{attribute 'GeneratedUsingTerminal: EL3773-0000-0019'}
{attribute addProperty BoxType "EL3773-0000-0019"}
{attribute addProperty Id "U2_SamplesAT %I*U2_Samples_2549228720"}
{attribute addProperty CRC "1977103279"}
{attribute addProperty Size "20"}
TYPE L2_Voltage_Samples_75D833AF :
STRUCT
	{attribute addProperty Name "U2_Samples"}
	U2_Samples AT %I* : U2_Samples_25492287;
END_STRUCT
END_TYPE

(* stored: Version 1.2.0.0, ProductVersion 3.1.4024.9
   DUT L2_Voltage_Samples_75D833AF: Id {fed5e55a-89fe-4a11-9afb-b5762e18c7ef} *)
